// A single structured metric attribute — a key/value label attached to a metric data point.
TYPE MetricAttribute :
STRUCT
	key : STRING(31);
	value : STRING(63);
END_STRUCT
END_TYPE

(* stored: Version 1.1.0.1
   DUT MetricAttribute: Id {2b8deae3-c8a3-4bbb-a37e-45bbb04ec461} *)
